// TIA Portal V20 export
TYPE "LER_typeStatusEm6"
// stored: Access Published
   STRUCT
      finalRollerCamEnabled : Bool;
      mandrelAnodeFrontYCamEnabled : Bool;
      mandrelAnodeFrontZCamEnabled : Bool;
      mandrelAnodeRearYCamEnabled : Bool;
      mandrelAnodeRearZCamEnabled : Bool;
      mandrelCathodeFrontYCamEnabled : Bool;
      mandrelCathodeFrontZCamEnabled : Bool;
      mandrelCathodeRearYCamEnabled : Bool;
      mandrelCathodeRearZCamEnabled : Bool;
      finalRollerMove : Bool;
      finalRollerMoveComplete : Bool;
      anodeGripComplete1 : Bool;
      anodeGripComplete2 : Bool;
      anodeGripComplete3 : Bool;
      cathodeGripComplete1 : Bool;
      cathodeGripComplete2 : Bool;
      cathodeGripComplete3 : Bool;
      finalRollerAnodePos : Bool;
      finalRollerCathodePos : Bool;
      stackStart : Bool;
      stackComplete : Bool;
      stackUpComplete : Bool;
      stackUngripComplete : Bool;
      stackGripComplete : Bool;
      onlyStackComplete : Bool;
      dancerHigh1 : Bool;
      dancerHigh2 : Bool;
      dancerHigh3 : Bool;
      dancerHigh4 : Bool;
      dancerLow1 : Bool;
      dancerLow2 : Bool;
      dancerLow3 : Bool;
      dancerLow4 : Bool;
      stopRequest : Bool;
      stopComplete : Bool;
      anodeSupplyRequest1 : Bool;
      anodeSupplyRequest2 : Bool;
      anodeFinishRequest : Bool;
      anodeSupplyCompleteCheck1 : Bool;
      anodeSupplyCompleteCheck2 : Bool;
      anodeFinishCompleteCheck : Bool;
      cathodeSupplyRequest1 : Bool;
      cathodeSupplyRequest2 : Bool;
      cathodeFinishRequest : Bool;
      cathodeSupplyCompleteCheck1 : Bool;
      cathodeSupplyCompleteCheck2 : Bool;
      cathodeFinishCompleteCheck : Bool;
      startCountCheck : DInt;
      finalRollerStart : LReal := 0.0;
      finalRollerEnd : LReal := 75.0;
      finalRollerDistance : LReal;
      mandrelBwdStartPos : LReal := 75.0;
      mandrelBwdEndPos : LReal := 82.5;
      mandrelFwdStartPos : LReal := 82.5;
      mandrelFwdEndPos : LReal := 90.0;
      mandrelUpStartPos : LReal := 75.0;
      mandrelUpEndPos : LReal := 82.5;
      mandrelDownStartPos : LReal := 87.0;
      mandrelDownEndPos : LReal := 90.0;
      outputCamOffset : LReal := 10.0;
      visionPosOffset : LReal := 0.0;
      visionTime : LReal := 50.0;
   END_STRUCT;
END_TYPE
